Staubli VAL3: MoveId.pjx

--- MoveId.pjx ---
Parameters version=s7.9 stackSize=5000 millimeterUnit=true
Program file=SameInstruct.pgx
Program file=start.pgx
Program file=stop.pgx
Data file=MoveId.dtx

--- MoveId.dtx ---
mdesc mNomSpeed
jointRx jJ
mdesc mMdesc
tool tTool = {fatherId=flange[0], ioLink=valve1}

--- start.pgx ---
program start()
begin

  call SameInstruct()


end
